{attribute 'qualified_only'}
VAR_GLOBAL
	nSpeed		: INT;
	bEnable		: BOOL;
	arValues	: ARRAY[0..9] OF INT;
END_VAR

(* stored: Version 1.1.0.1, ProductVersion 3.1.4024.12
   GVL GVL_Hmi: Id {f5f523de-3785-4f7b-a814-dd5df81cfa6b} *)
